// TwinCAT 3 PLC project StatePatternPlc
// ProgramVersion: 3.1.4023.0
// libraries:
//   Tc2_Standard, * (Beckhoff Automation GmbH)
//   Tc2_System, * (Beckhoff Automation GmbH)
//   Tc2_XmlDataSrv, * (Beckhoff Automation GmbH)
//   Tc3_EventLogger, * (Beckhoff Automation GmbH)
//   Tc3_Module, * (Beckhoff Automation GmbH)
// project tree:
//   02_Machine/01_States/ FB_StateEStop.TcPOU, FB_StateBegin.TcPOU, FB_StateInit.TcPOU, FB_StateReadParameters.TcPOU, FB_StateError.TcPOU
//   02_Machine/ FB_MainStateMachine.TcPOU, I_State.TcIO, ST_MainStateMachineHmi.TcDUT, ST_MainStateMachineHmiCommand.TcDUT, ST_MainStateMachineHmiStatus.TcDUT
//   03_IO/ IO.TcGVL
//   04_Safety/ Safety.TcGVL
//   05_MachineParameters/ MachineParameters.TcGVL, ST_MachineParameters.TcDUT, ST_MachineParametersAxis.TcDUT
//   06_Hmi/ Hmi.TcGVL
//   / PlcTask.TcTTO
//   01_Main/ MAIN.TcPOU
// real-time tasks:
//   TASK PlcTask: cycle T#10ms, priority 6, ADS port 350

CONFIGURATION StatePatternPlc
    RESOURCE PLC ON TwinCAT3
        TASK PlcTask(INTERVAL := T#10ms, PRIORITY := 6);
        PROGRAM MAIN WITH PlcTask : MAIN;
    END_RESOURCE
END_CONFIGURATION

// ---- 02_Machine/ST_MainStateMachineHmi.TcDUT
TYPE ST_MainStateMachineHmi :
STRUCT
	stCommand				: ST_MainStateMachineHmiCommand;
	stStatus				: ST_MainStateMachineHmiStatus;
END_STRUCT
END_TYPE

// ---- 02_Machine/ST_MainStateMachineHmiCommand.TcDUT
TYPE ST_MainStateMachineHmiCommand :
STRUCT
	bStartButton				: BOOL;
	bStopButton					: BOOL;
END_STRUCT
END_TYPE

// ---- 02_Machine/ST_MainStateMachineHmiStatus.TcDUT
TYPE ST_MainStateMachineHmiStatus :
STRUCT
	sActState					: STRING;
END_STRUCT
END_TYPE

// ---- 05_MachineParameters/ST_MachineParameters.TcDUT
TYPE ST_MachineParameters :
STRUCT
	sSerialNumber			: STRING;
	stAxisM1				: ST_MachineParametersAxis;
	stAxisM2				: ST_MachineParametersAxis;
END_STRUCT
END_TYPE

// ---- 05_MachineParameters/ST_MachineParametersAxis.TcDUT
TYPE ST_MachineParametersAxis :
STRUCT
	fSoftPositionLimitMax			: LREAL;
	fSoftPositionLimitMin			: LREAL;
	fDefaultVelocity				: LREAL;
	fHomePosition					: LREAL;
END_STRUCT
END_TYPE

// ---- 03_IO/IO.TcGVL
{attribute 'qualified_only'}
VAR_GLOBAL
	bStartButton			: BOOL;
	bStopButton				: BOOL;
END_VAR

// ---- 04_Safety/Safety.TcGVL
{attribute 'qualified_only'}
VAR_GLOBAL
	bEStopOK			: BOOL;
END_VAR

// ---- 05_MachineParameters/MachineParameters.TcGVL
{attribute 'qualified_only'}
VAR_GLOBAL
	sFilePath			: STRING := 'C:\Temp\MachineParameters.xml';
	sXPath				: STRING := '/MachineParameters/Data';
	stData				: ST_MachineParameters;
END_VAR

// ---- 06_Hmi/Hmi.TcGVL
{attribute 'qualified_only'}
VAR_GLOBAL
	stMainStateMachine				: ST_MainStateMachineHmi;
END_VAR

// ---- 02_Machine/I_State.TcIO
INTERFACE I_State

METHOD SafetyAcknowledged
VAR_INPUT
END_VAR
END_METHOD

METHOD StopButtonPressed
END_METHOD

METHOD ClearErrors
END_METHOD

METHOD GetDescription : STRING
END_METHOD

METHOD Execute
END_METHOD

METHOD StartButtonPressed
END_METHOD

METHOD SafetyTripped
VAR_INPUT
END_VAR
END_METHOD

END_INTERFACE

// ---- 01_Main/MAIN.TcPOU
PROGRAM MAIN
VAR
	fbMainStateMachine			: FB_MainStateMachine(
		stHmi						:= Hmi.stMainStateMachine);
END_VAR

fbMainStateMachine.Execute();

END_PROGRAM

// ---- 02_Machine/FB_MainStateMachine.TcPOU
FUNCTION_BLOCK FB_MainStateMachine
VAR
	_fbStateBegin				: FB_StateBegin(
		fbMainStateMachine			:= THIS^);
	_fbStateReadParameters		: FB_StateReadParameters(
		fbMainStateMachine			:= THIS^);
	_fbStateEStop				: FB_StateEStop(
		fbMainStateMachine			:= THIS^);
	_fbStateInit				: FB_StateInit(
		fbMainStateMachine			:= THIS^);
	_fbStateError				: FB_StateError(
		fbMainStateMachine			:= THIS^);
	_ipActState					: I_State := _fbStateBegin;
	_ipPrevState				: I_State := _fbStateBegin;
	_fbTcMessage				: FB_TcMessage;
	_refHmi						: REFERENCE TO ST_MainStateMachineHmi;
END_VAR

PROPERTY ipStateError : I_State
GET
ipStateError := _fbStateError;
END_GET
END_PROPERTY

PROPERTY ipStateEStop : I_State
GET
ipStateEStop := _fbStateEStop;
END_GET
END_PROPERTY

METHOD Execute
VAR_INST
	_fbFTrigStartButton			: F_TRIG;
	_fbFTrigStopButton			: F_TRIG;
	_fbFTrigEStopOK				: F_TRIG;
	_fbRTrigEStopOK				: R_TRIG;
END_VAR
_fbFTrigStartButton(CLK := _refHmi.stCommand.bStartButton);

_ipActState.Execute();

IF _fbFTrigStartButton.Q THEN
	_ipActState.StartButtonPressed();
END_IF

_fbFTrigStopButton(CLK := _refHmi.stCommand.bStopButton);

IF _fbFTrigStopButton.Q THEN
	_ipActState.StopButtonPressed();
END_IF

_fbFTrigEStopOK(CLK := Safety.bEStopOK);

IF _fbFTrigEStopOK.Q THEN
	_ipActState.SafetyTripped();
END_IF

_fbRTrigEStopOK(CLK := Safety.bEStopOK);

IF _fbRTrigEStopOK.Q THEN
	_ipActState.SafetyAcknowledged();
END_IF

_refHmi.stStatus.sActState := _ipActState.GetDescription();
END_METHOD

PROPERTY ipStateInit : I_State
GET
ipStateInit := _fbStateInit;
END_GET
END_PROPERTY

METHOD SetState
VAR_INPUT
	ipNextState			: I_State;
END_VAR
VAR
	sTemp				: STRING;
END_VAR
_ipPrevState := _ipActState;
_ipActState := ipNextState;
sTemp := _ipActState.GetDescription();
_fbTcMessage.ipArguments.Clear().AddString(sTemp);
_fbTcMessage.Send(0);
END_METHOD

METHOD FB_init : BOOL
VAR_INPUT
	// if TRUE, the retain variables are initialized (warm start / cold start)
	bInitRetains			: BOOL;
	// if TRUE, the instance afterwards gets moved into the copy code (online
	// change)
	bInCopyCode				: BOOL;
	stHmi					: REFERENCE TO ST_MainStateMachineHmi;
END_VAR
_refHmi REF= stHmi;

_fbTcMessage.CreateEx(
	stEventEntry	:= TC_EVENTS.StatePatternEvents.Info010StateChanged,
	ipSourceInfo	:= 0);
END_METHOD

PROPERTY ipPrevState : I_State
GET
ipPrevState := _ipPrevState;
END_GET
END_PROPERTY

PROPERTY ipStateReadParameters : I_State
GET
ipStateReadParameters := _fbStateReadParameters;
END_GET
END_PROPERTY

END_FUNCTION_BLOCK

// ---- 02_Machine/01_States/FB_StateBegin.TcPOU
FUNCTION_BLOCK FB_StateBegin IMPLEMENTS I_State
VAR
	_refMainStateMachine		: REFERENCE TO FB_MainStateMachine;
	_fbTcMessage				: FB_TcMessage;
	_fbTon						: TON;
END_VAR

METHOD SafetyTripped
VAR_INPUT
END_VAR
END_METHOD

METHOD FB_init : BOOL
VAR_INPUT
	// if TRUE, the retain variables are initialized (warm start / cold start)
	bInitRetains			: BOOL;
	// if TRUE, the instance afterwards gets moved into the copy code (online
	// change)
	bInCopyCode				: BOOL;
	fbMainStateMachine		: REFERENCE TO FB_MainStateMachine;
END_VAR
_refMainStateMachine REF= fbMainStateMachine;
_fbTcMessage.CreateEx(
	stEventEntry	:= TC_EVENTS.StatePatternEvents.Info001MachineStarted,
	ipSourceInfo	:= 0);
END_METHOD

METHOD SafetyAcknowledged
VAR_INPUT
END_VAR
END_METHOD

METHOD ClearErrors
END_METHOD

METHOD StartButtonPressed
END_METHOD

METHOD GetDescription : STRING
GetDescription := 'Begin';
END_METHOD

METHOD Execute
IF _TaskInfo[GETCURTASKINDEXEX()].FirstCycle THEN
	_fbTcMessage.Send(0);
END_IF

_fbTon(IN := TRUE, PT := T#100MS);

IF _fbTon.Q THEN
	_fbTon(IN := FALSE);
	_refMainStateMachine.SetState(_refMainStateMachine.ipStateReadParameters);
END_IF
END_METHOD

METHOD StopButtonPressed
END_METHOD

END_FUNCTION_BLOCK

// ---- 02_Machine/01_States/FB_StateReadParameters.TcPOU
FUNCTION_BLOCK FB_StateReadParameters IMPLEMENTS I_State
VAR
	_refMainStateMachine		: REFERENCE TO FB_MainStateMachine;
	_fbXmlSrvRead				: FB_XmlSrvRead;
	_fbTcAlarm					: FB_TcAlarm;
END_VAR

METHOD GetDescription : STRING
GetDescription := 'Read parameters';
END_METHOD

METHOD ClearErrors
_fbTcAlarm.Clear(
	nTimeStamp			:= 0,
	bResetConfirmation	:= TRUE);
END_METHOD

METHOD StopButtonPressed
END_METHOD

METHOD StartButtonPressed
END_METHOD

METHOD Execute
_fbXmlSrvRead(
	pSymAddr	:= ADR(MachineParameters.stData),
	cbSymSize	:= SIZEOF(MachineParameters.stData),
	sFilePath	:= MachineParameters.sFilePath,
	sXPath		:= MachineParameters.sXPath,
	bExecute	:= TRUE);

IF NOT _fbXmlSrvRead.bBusy AND NOT _fbXmlSrvRead.bError THEN
	_fbXmlSrvRead(bExecute := FALSE);
	_refMainStateMachine.SetState(_refMainStateMachine.ipStateEStop);
ELSIF NOT _fbXmlSrvRead.bBusy AND _fbXmlSrvRead.bError THEN
	_fbTcAlarm.ipArguments.Clear().AddUDInt(_fbXmlSrvRead.nErrId);
	_fbTcAlarm.Raise(0);
	_fbXmlSrvRead(bExecute := FALSE);
	_refMainStateMachine.SetState(_refMainStateMachine.ipStateError);
END_IF
END_METHOD

METHOD FB_init : BOOL
VAR_INPUT
	// if TRUE, the retain variables are initialized (warm start / cold start)
	bInitRetains			: BOOL;
	// if TRUE, the instance afterwards gets moved into the copy code (online
	// change)
	bInCopyCode				: BOOL;
	fbMainStateMachine		: REFERENCE TO FB_MainStateMachine;
END_VAR
_refMainStateMachine REF= fbMainStateMachine;
_fbTcAlarm.CreateEx(
	stEventEntry		:= TC_EVENTS.StatePatternEvents.Error100ParameterReadError,
	bWithConfirmation	:= FALSE,
	ipSourceInfo		:= 0);
END_METHOD

METHOD SafetyTripped
END_METHOD

METHOD SafetyAcknowledged
END_METHOD

END_FUNCTION_BLOCK

// ---- 02_Machine/01_States/FB_StateEStop.TcPOU
FUNCTION_BLOCK FB_StateEStop IMPLEMENTS I_State
VAR
	_refMainStateMachine		: REFERENCE TO FB_MainStateMachine;
END_VAR

METHOD StopButtonPressed
END_METHOD

METHOD StartButtonPressed
END_METHOD

METHOD FB_init : BOOL
VAR_INPUT
	// if TRUE, the retain variables are initialized (warm start / cold start)
	bInitRetains			: BOOL;
	// if TRUE, the instance afterwards gets moved into the copy code (online
	// change)
	bInCopyCode				: BOOL;
	fbMainStateMachine		: REFERENCE TO FB_MainStateMachine;
END_VAR
_refMainStateMachine REF= fbMainStateMachine;
END_METHOD

METHOD SafetyAcknowledged
VAR_INPUT
END_VAR
_refMainStateMachine.SetState(_refMainStateMachine.ipStateInit);
END_METHOD

METHOD ClearErrors
END_METHOD

METHOD Execute
END_METHOD

METHOD GetDescription : STRING
GetDescription := 'Emergency stop';
END_METHOD

METHOD SafetyTripped
VAR_INPUT
END_VAR
END_METHOD

END_FUNCTION_BLOCK

// ---- 02_Machine/01_States/FB_StateInit.TcPOU
FUNCTION_BLOCK FB_StateInit IMPLEMENTS I_State
VAR
	_refMainStateMachine		: REFERENCE TO FB_MainStateMachine;
END_VAR

METHOD StartButtonPressed
END_METHOD

METHOD StopButtonPressed
END_METHOD

METHOD SafetyAcknowledged
VAR_INPUT
END_VAR
END_METHOD

METHOD ClearErrors
END_METHOD

METHOD SafetyTripped
VAR_INPUT
END_VAR
_refMainStateMachine.SetState(_refMainStateMachine.ipStateEStop);
END_METHOD

METHOD FB_init : BOOL
VAR_INPUT
	// if TRUE, the retain variables are initialized (warm start / cold start)
	bInitRetains			: BOOL;
	// if TRUE, the instance afterwards gets moved into the copy code (online
	// change)
	bInCopyCode				: BOOL;
	fbMainStateMachine		: REFERENCE TO FB_MainStateMachine;
END_VAR
_refMainStateMachine REF= fbMainStateMachine;
END_METHOD

METHOD GetDescription : STRING
GetDescription := 'Initialization';
END_METHOD

METHOD Execute
END_METHOD

END_FUNCTION_BLOCK

// ---- 02_Machine/01_States/FB_StateError.TcPOU
FUNCTION_BLOCK FB_StateError IMPLEMENTS I_State
VAR
	_refMainStateMachine		: REFERENCE TO FB_MainStateMachine;
	_fbXmlSrvRead				: FB_XmlSrvRead;
	_nErrorAckCount				: UDINT;
END_VAR

METHOD FB_init : BOOL
VAR_INPUT
	// if TRUE, the retain variables are initialized (warm start / cold start)
	bInitRetains			: BOOL;
	// if TRUE, the instance afterwards gets moved into the copy code (online
	// change)
	bInCopyCode				: BOOL;
	fbMainStateMachine		: REFERENCE TO FB_MainStateMachine;
END_VAR
_refMainStateMachine REF= fbMainStateMachine;
END_METHOD

METHOD StopButtonPressed
END_METHOD

METHOD Execute
END_METHOD

METHOD SafetyTripped
END_METHOD

METHOD ClearErrors
END_METHOD

METHOD SafetyAcknowledged
END_METHOD

METHOD GetDescription : STRING
GetDescription := 'Error';
END_METHOD

METHOD StartButtonPressed
IF _refMainStateMachine.ipPrevState <> 0 THEN
	_nErrorAckCount := _nErrorAckCount + 1;
	_refMainStateMachine.ipPrevState.ClearErrors();
	_refMainStateMachine.SetState(_refMainStateMachine.ipPrevState);
END_IF
END_METHOD

END_FUNCTION_BLOCK
